FUNCTION_BLOCK ABSTRACT TaskBase EXTENDS CyclicBase IMPLEMENTS I_Task
VAR
	_Busy : BOOL;
	_Error : BOOL;
	_Done : BOOL;
	State: INT;
END_VAR

{analysis -2}

PROPERTY Busy : BOOL
GET
Busy := _Busy;
END_GET
END_PROPERTY

PROPERTY Done : BOOL
GET
Done := _Done;
END_GET
END_PROPERTY

PROPERTY Error : BOOL
GET
Error := _Error;
END_GET
END_PROPERTY

END_FUNCTION_BLOCK

(* stored: Version 1.1.0.1
   POU TaskBase: Id {1c339505-1708-4516-99c7-fe794eeac80e}, SpecialFunc None
   Property Busy: Id {c2084324-8459-4ee4-a5af-e278c120f558}
   Get Get: Id {d282fb96-d58b-4810-8232-8142176d20dd}
   Property Done: Id {8c6a969e-0897-4aef-ae58-391d7d66beb9}
   Get Get: Id {18a849d4-6a1c-4e5f-9c47-5214e6aa579c}
   Property Error: Id {45193d04-4a27-4fd3-921b-d8f6914de5c2}
   Get Get: Id {8a0917a7-f9f5-4823-9a91-98c67cd20cc9} *)
